FUNCTION_BLOCK SERVER_0_3 (* 3 RD/0 SD Server Interface *)
  (* Standard: 61499-1; Classification: Communications *)
  (* Version 0.0, 2003-05-14, JHC, Rockwell Automation *)
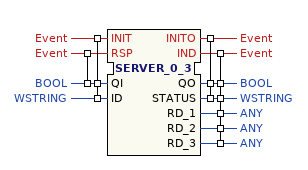
  EVENT_INPUT
    INIT WITH QI, ID;
    RSP WITH QI;
  END_EVENT
  EVENT_OUTPUT
    INITO WITH QO, STATUS;
    IND WITH QO, STATUS, RD_1, RD_2, RD_3;
  END_EVENT
  VAR_INPUT
    QI : BOOL;
    ID : WSTRING;
  END_VAR
  VAR_OUTPUT
    QO : BOOL;
    STATUS : WSTRING;
    RD_1 : ANY;
    RD_2 : ANY;
    RD_3 : ANY;
  END_VAR
END_FUNCTION_BLOCK
